(* CODESYS project Uppgift 8.project

Project tree, tasks and I/O mapping:
  Device : CODESYS Control Win V3, 3S - Smart Software Solutions GmbH, order no. 305021, version 3.5.10.40
    application Application
      libraries: Standard, * (System)
      task MainTask (cyclic, interval t#20ms, priority 1) calls PLC_PRG
      task VISU_TASK (cyclic, interval 100 ms, priority 31) calls VisuElems.Visu_Prg
      program PLC_PRG [LD]
      global variables GVL
      visualisation Visualization
  libraries: VisuSymbols, 3.5.10.0 (System)
  text list GlobalTextList
*)

// Device/Application/GVL
{attribute 'qualified_only'}
VAR_GLOBAL
	CTU_0: CTU;
	Lamp_Green: BOOL;
	Btn_2: BOOL;
	Btn_1: BOOL;
	Cunter_Up: WORD;
	CounterToReset: WORD;
	CTU_1: CTu;
	Returnvalue: BOOL;
END_VAR

// Device/Application/PLC_PRG
PROGRAM PLC_PRG
VAR
	CTU_0: CTU;
	Lamp_Green: BOOL;
	Btn_2: BOOL;
	Btn_1: BOOL;
	Cunter_Up: WORD;
	CounterToReset: WORD;
	CTU_1: CTu;
	Returnvalue: BOOL;
END_VAR

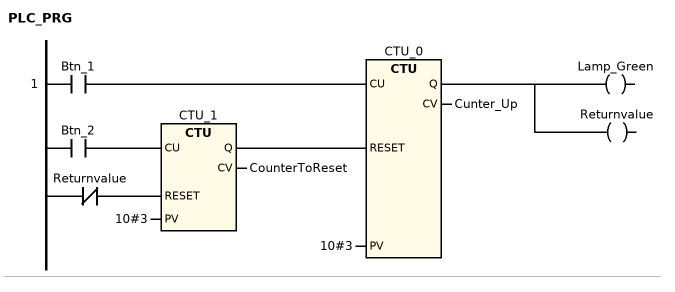
// NETWORK 1
CTU_1(CU := Btn_2, RESET := NOT Returnvalue, PV := 10#3, CV => CounterToReset); // CTU
CTU_0(CU := Btn_1, RESET := CTU_1.Q, PV := 10#3, CV => Cunter_Up); // CTU
Lamp_Green := CTU_0.Q;
Returnvalue := CTU_0.Q;

END_PROGRAM

// Device/Application/Visualization
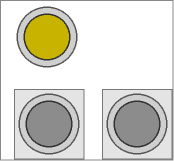
VISUALIZATION Visualization  // 174x161
    Lamp1 (12,2 70x70), variable: GVL.Lamp_Green, style: Lamp-Lamp1-Yellow
    PushSwitch (14,89 70x70), variable: GVL.Btn_1, behaviour: TOGGLE, style: Switch-PushSwitch-Gray
    PushSwitch (102,89 70x70), variable: GVL.Btn_2, behaviour: TOGGLE, style: Switch-PushSwitch-Gray
END_VISUALIZATION
